// TIA Portal V16 export
// export: Created 2023-01-03T15:35:06.522745Z, ExportSetting WithDefaults, DisplayName Totally Integrated Automation Portal, DisplayVersion V16, DisplayName TIA Portal Version Control Interface, DisplayVersion V16, DisplayName TIA Portal Openness, DisplayVersion V16, DisplayName STEP 7 Professional, DisplayVersion V16, DisplayName STEP 7 Safety, DisplayVersion V16, DisplayName WinCC Advanced, DisplayVersion V16
FUNCTION "CYLINDER_MANUAL" : Void   // FC2, LAD
{ S7_Optimized_Access := 'TRUE' }
VERSION : 0.1
// stored: AutoNumber true, IsIECCheckEnabled false, SetENOAutomatically false, UDAEnableTagReadback false
   VAR_INPUT
      "MANUAL M4 RETRACT  PB" : Bool;
      "MANUAL M4 EXTEND  PB" : Bool;
      EXTENDED : Bool;
      RETRACTED : Bool;
   END_VAR
   VAR_OUTPUT
      "M4 EXTEND" : Bool;
      "M4 RETRACT" : Bool;
      "EXTEND INDICATION" : Bool;
      "RETRACT INDICATION" : Bool;
   END_VAR
BEGIN

REGION Network 1: EXTEND THE CYLINDER
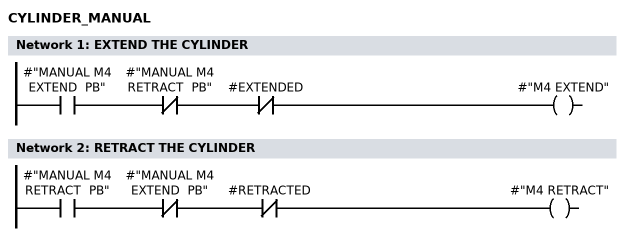
   RUNG wire#powerrail
      Contact( #"MANUAL M4 EXTEND  PB" )
      I_Contact( #"MANUAL M4 RETRACT  PB" )
      I_Contact( #EXTENDED )
      Coil( #"M4 EXTEND" )
   END_RUNG
   // the same network as SCL:
   #"M4 EXTEND" := #"MANUAL M4 EXTEND  PB" AND NOT #"MANUAL M4 RETRACT  PB" AND NOT #EXTENDED;
END_REGION

REGION Network 2: RETRACT THE CYLINDER
   RUNG wire#powerrail
      Contact( #"MANUAL M4 RETRACT  PB" )
      I_Contact( #"MANUAL M4 EXTEND  PB" )
      I_Contact( #RETRACTED )
      Coil( #"M4 RETRACT" )
   END_RUNG
   // the same network as SCL:
   #"M4 RETRACT" := #"MANUAL M4 RETRACT  PB" AND NOT #"MANUAL M4 EXTEND  PB" AND NOT #RETRACTED;
END_REGION
END_FUNCTION
